// TIA Portal V15.1 export
// export: Created 2024-06-21T08:41:11.7046942Z, ExportSetting WithDefaults, DisplayName Totally Integrated Automation Portal, DisplayVersion V15.1 Update 5, DisplayName TIA Portal Openness, DisplayVersion V15.1 Update 5, DisplayName SINAMICS Startdrive Advanced, DisplayVersion V15.1, DisplayName G130, G150, S120, S150, SINAMICS MV, S210, DisplayVersion V15.1, DisplayName G110M, G120, G120C, G120D, G120P, DisplayVersion V15.1, DisplayName STEP 7 Professional, DisplayVersion V15.1 Update 5, DisplayName STEP 7 Safety, DisplayVersion V15.1, DisplayName WinCC Professional, DisplayVersion V15.1 Update 5, DisplayName SIMATIC Visualization Architect, DisplayVersion V15.1
FUNCTION "LGBCalcRampMoviDrive" : Void   // FC6629, SCL
{ S7_Optimized_Access := 'TRUE' }
VERSION : 0.1
// stored: AutoNumber false, IsIECCheckEnabled false, SetENOAutomatically False, UDAEnableTagReadback false
   VAR_INPUT
      I_Ramp : Time;   // Ramp send in miliseconds (range : 100-10000ms, if 0 then default 1s will be used)
      I_SetpointSpeed : Real;   // Speed value 0-100% / High speed value 0-100%
      C_MotorRPM : Real;   // Reference RPM of the motor
      C_RatioGearbox : Real;   // Ratio Gearbox <-> Motor
      C_Diameter : Real;   // Diameter in mm
      C_Acceleration : Real;   // Acceleration in m/s²
   END_VAR
   VAR_OUTPUT
      O_RampToDrive : DInt;   // Ramp to Drive in millisec
      H_RampToDrive : DInt;   // Ramp to Drive in millisec
      H_Ramp : DInt;   // Ramp in millisec
      "H_m/min" : Real;   // Speed in m/min
      "H_m/sec" : Real;   // Speed in m/sec
      H_Acceleration : Real;   // Acceleration in m/s²
   END_VAR
   VAR_TEMP
      SetpointSpeed : Real;   // Speed value 0-100% / High speed value 0-100%
      RampToDrive : DInt;   // Ramp to Drive in millisec
      Ramp : DInt;   // Ramp in millisec
      "m/min" : Real;   // Speed in m/min
      "m/sec" : Real;   // Speed in m/sec
   END_VAR
BEGIN
   // LOGIC
   IF (#I_SetpointSpeed <> 0.0) AND (#C_MotorRPM <> 0.0) AND (#C_RatioGearbox <> 0.0) AND (#C_Diameter <> 0.0) AND (#C_Acceleration <> 0.0) THEN
       IF (#I_SetpointSpeed > 0.0) THEN
           #SetpointSpeed := #I_SetpointSpeed;
       ELSE
           #SetpointSpeed := #I_SetpointSpeed * -1.0;
       END_IF;

       // v = 2 * Pi * r * n [m/min] 
       #"m/min" := 2 * 3.141592653 * ((#C_Diameter / 2) / 1000) * (((#SetpointSpeed / 100.0) * #C_MotorRPM) / #C_RatioGearbox);

       // v [m/sec] 
       #"m/sec" := #"m/min" / 60;

       // Ramp
       #RampToDrive := REAL_TO_DINT(((#"m/sec" / #C_Acceleration) * (3000 / ((#SetpointSpeed / 100.0) * #C_MotorRPM)) * 1000));
       #Ramp := REAL_TO_DINT((#"m/sec" / #C_Acceleration) * 1000);
   ELSE
       #"m/min" := 0.0;
       #"m/sec" := 0.0;
       #RampToDrive := 0;
       #Ramp := T#0s;
   END_IF;

   IF NOT ((#C_MotorRPM <> 0.0) AND (#C_RatioGearbox <> 0.0) AND (#C_Diameter <> 0.0) AND (#C_Acceleration <> 0.0)) THEN
       #RampToDrive := #I_Ramp;
   END_IF;

   // OUTPUTS
   #O_RampToDrive := #RampToDrive;
   #H_RampToDrive := #RampToDrive;
   #H_Ramp := #Ramp;
   #"H_m/min" := #"m/min";
   #"H_m/sec" := #"m/sec";
   #H_Acceleration := #C_Acceleration;
END_FUNCTION
